// SIMATIC S7-200 project (STEP 7-Micro/WIN), CPU 224XP CN REL 02.01

ORGANIZATION_BLOCK MAIN:OB1
TITLE= 
// PROGRAM COMMENTS
// Press F1 for help and example program
//  
BEGIN
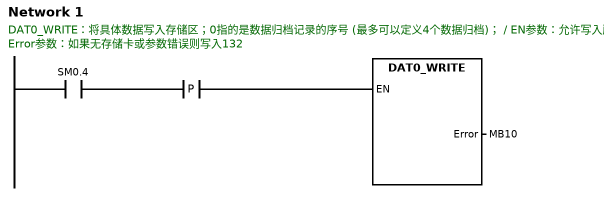
Network 1
// DAT0_WRITE：将具体数据写入存储区；0指的是数据归档记录的序号 (最多可以定义4个数据归档)；
// EN参数：允许写入所选的数据归档记录事件触发(不要每个扫描周期都写，最大100,000个周期)
// Error参数：如果无存储卡或参数错误则写入132
LD     SM0.4
EU
CALL   DAT0_WRITE:SBR1, MB10
END_ORGANIZATION_BLOCK

// SBR1: protected block, not included

// (further data pages could not be read)
